FUNCTION FC_BOOLARR_TO_BYTE
VAR_INPUT
	pMyByte : POINTER TO BYTE; // Destination  
	pMyBool : POINTER TO BOOL; // Source   
	nSize	: UINT;               
END_VAR
VAR
    i : UINT;                       
	myByte :  BYTE; 
END_VAR

FOR i:= 0 TO nSize-1 BY 8 DO
	myByte := FC_BOOLBYTE_TO_BYTE(ADR(pMyBool[i]));
	MEMCPY(ADR(pMyByte[i/8]), ADR(myByte), SIZEOF(BYTE));
END_FOR

END_FUNCTION

(* stored: Version 1.1.0.1, ProductVersion 3.1.4024.13
   POU FC_BOOLARR_TO_BYTE: Id {f8c33bda-ceee-4eb4-9180-eed54a304c16}, SpecialFunc None *)
